FUNCTION_BLOCK XCBR_Circuit_Breaker_SIMULATION (* Composite Function Block Type *)
  (* Standard: 61499-2 *)
  (* Version 0.0, 12/11/2023, Cheyan, Schneider Electric, template *)
  PACKAGE Main;
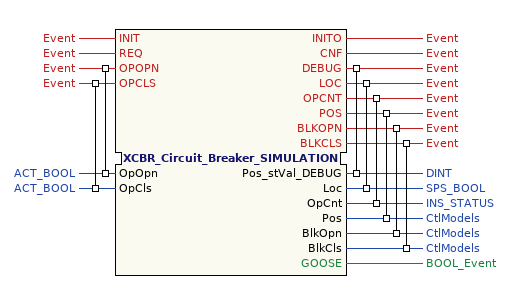
  EVENT_INPUT
    INIT; (* Initialization Request *)
    REQ; (* Normal Execution Request *)
    OPOPN WITH OpOpn;
    OPCLS WITH OpCls;
  END_EVENT
  EVENT_OUTPUT
    INITO; (* Initialization Confirm *)
    CNF; (* Execution Confirmation *)
    DEBUG WITH Pos_stVal_DEBUG;
    LOC WITH Loc;
    OPCNT WITH OpCnt;
    POS WITH Pos;
    BLKOPN WITH BlkOpn;
    BLKCLS WITH BlkCls;
  END_EVENT
  VAR_INPUT
    OpOpn : ACT_BOOL; (* Input event qualifier *)
    OpCls : ACT_BOOL;
  END_VAR
  VAR_OUTPUT
    Pos_stVal_DEBUG : DINT;
    Loc : SPS_BOOL;
    OpCnt : INS_STATUS;
    Pos : CtlModels;
    BlkOpn : CtlModels;
    BlkCls : CtlModels;
  END_VAR
  PLUGS
    GOOSE : BOOL_Event;
  END_PLUGS
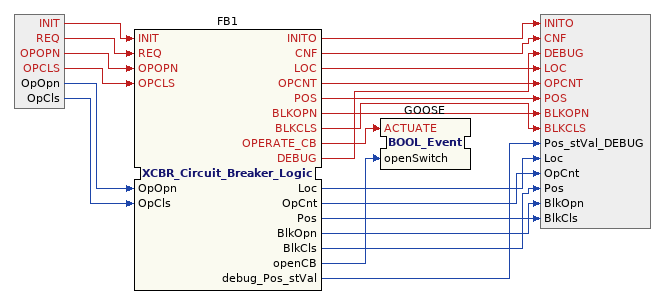
  FBS
    FB1 : XCBR_Circuit_Breaker_Logic;
  END_FBS
  EVENT_CONNECTIONS
    INIT TO FB1.INIT;
    REQ TO FB1.REQ;
    FB1.INITO TO INITO;
    FB1.CNF TO CNF;
    FB1.OPERATE_CB TO GOOSE.ACTUATE;
    FB1.DEBUG TO DEBUG;
    FB1.LOC TO LOC;
    FB1.OPCNT TO OPCNT;
    FB1.POS TO POS;
    FB1.BLKOPN TO BLKOPN;
    FB1.BLKCLS TO BLKCLS;
    OPOPN TO FB1.OPOPN;
    OPCLS TO FB1.OPCLS;
  END_CONNECTIONS
  DATA_CONNECTIONS
    FB1.openCB TO GOOSE.openSwitch;
    FB1.debug_Pos_stVal TO Pos_stVal_DEBUG;
    FB1.Loc TO Loc;
    FB1.OpCnt TO OpCnt;
    FB1.Pos TO Pos;
    FB1.BlkOpn TO BlkOpn;
    FB1.BlkCls TO BlkCls;
    OpOpn TO FB1.OpOpn;
    OpCls TO FB1.OpCls;
  END_CONNECTIONS
END_FUNCTION_BLOCK
